Fanuc KAREL source: kt00644.KL

-- PROVISIONAL review KL for V1013-1; original PC SHA256 e1b4a1370d9cffa532d57e57cbbdfda6e969248b25e8500a416a2d44073d4770
-- Incomplete behavior may be omitted. Consult companion uncertainty JSON. Do not deploy.
PROGRAM KT00644
%NOLOCKGROUP
VAR
  OUT : REAL
-- UNRESOLVED_DECL H1 type=002017
-- UNRESOLVED_DECL H2 type=002017
BEGIN
  -- UNRESOLVED_PC offsets 5-19; opcodes 2E,22,9D,33,B4
  -- UNRESOLVED_PC offsets 24-38; opcodes 2E,22,9D,33,B4
  -- UNRESOLVED_PC offsets 43-57; opcodes 2E,22,9D,33,B4
  -- UNRESOLVED_PC offsets 62-76; opcodes 2E,22,9D,33,B4
  -- UNRESOLVED_PC offsets 81-98; opcodes 22,9D,33,B3,48,64,23
  -- UNRESOLVED_PC offsets 103-107; opcodes 7F
END KT00644
